(* IEC 61131-3 sources: AXOpen/src/components.rexroth.drives/ctrl/src/AxoCtrlxDriveXsc/v_6_x_x (part 2) *)

                        AxoStop_Deceleration := 1000.0;         // mm/s2
                        AxoStop_Jerk := 150000.0;               // mm/s3
                        AxoHalt_Deceleration := 1000.0;         // mm/s2
                        AxoHalt_Jerk := 150000.0;               // mm/s3
                        AxoHome_Position := 0.0;                // mm
                        AxoHome_HommingMode := 615;             // Negative direction, travel range limit switch, negative edge (NC contact), no Home switch evaluation, no Reference mark evaluation
                        AxoHome_Velocity := 2.0;                // mm/s
                        AxoHome_Acceleration := 1000.0;         // mm/s2
                        AxoHome_Deceleration := 1000.0;         // mm/s2
                        AxoSetPosition_Position := 0.0;         // mm
                        AxoMoveAbsolute_Position := 0.0;        // mm
                        AxoMoveAbsolute_Velocity := 5.0;        // mm/s
                        AxoMoveAbsolute_Acceleration := 1000.0; // mm/s2
                        AxoMoveAbsolute_Deceleration := 1000.0; // mm/s2
                        AxoMoveAbsolute_Jerk := 150000.0;       // mm/s3
                        AxoMoveRelative_Distance := 5.0;        // mm
                        AxoMoveRelative_Velocity := 5.0;        // mm/s
                        AxoMoveRelative_Acceleration := 1000.0; // mm/s2
                        AxoMoveRelative_Deceleration := 1000.0; // mm/s2
                        AxoMoveRelative_Jerk := 150000.0;       // mm/s3
                        AxoMoveAdditive_Distance := 5.0;        // mm
                        AxoMoveAdditive_Velocity := 5.0;        // mm/s
                        AxoMoveAdditive_Acceleration := 1000.0; // mm/s2
                        AxoMoveAdditive_Deceleration := 1000.0; // mm/s2
                        AxoMoveAdditive_Jerk := 150000.0;       // mm/s3
                        AxoMoveVelocity_Velocity := 5.0;        // mm/s
                        AxoMoveVelocity_Acceleration := 1000.0; // mm/s2
                        AxoMoveVelocity_Deceleration := 1000.0; // mm/s2
                        AxoMoveVelocity_Jerk := 150000.0;       // mm/s3
                        AxoTorqueControl_Torque := 0.0;         // N
                        AxoTorqueControl_TorqueRamp := 1.0;     // N/s
                        AxoTorqueControl_Velocity := 5.0;       // mm/s
                        AxoTorqueControl_Acceleration := 1000.0;// mm/s2
                        AxoTorqueControl_Deceleration := 1000.0;// mm/s2
                        AxoTorqueControl_Jerk := 150000.0;      // mm/s3
                        AxoJog_Velocity := 2.0;                 // mm/s
                        AxoJog_Acceleration := 500.0;           // mm/s2
                        AxoJog_Deceleration := 500.0;           // mm/s2
                        AxoJog_Jerk := 150000.0;                // mm/s3
                        AxisRefExt.Outputs.BipolarTorqueLimitation_S_0_0092_0_0 := INT#1000;  // 1000~~ 100%
                    ELSIF AxisType = eAxoDriveAxisType#Rotary THEN
                        //  Position
                        ScalingConstantRequiredPosition     :=  TO_LREAL(_S_0_0079) / LREAL#360.0;
                        ScalingConstantActualPosition       :=  LREAL#1.0/ScalingConstantRequiredPosition;
                        //  Velocity
                        ScalingConstantRequiredVelocity     := _exp[-_S_0_0046] / (TO_LREAL(_S_0_0045));
                        ScalingConstantActualVelocity       := LREAL#1.0/ScalingConstantRequiredVelocity;
                        //  Acceleration
                        ScalingConstantRequiredAcceleration :=  _exp[-_S_0_0162] / (TO_LREAL(_S_0_0161) * LREAL#180.0 /System.Math.Constants#PI);
                        ScalingConstantActualAcceleration   := LREAL#1.0/ScalingConstantRequiredAcceleration;
                        //  Deceleration
                        ScalingConstantRequiredDeceleration := ScalingConstantRequiredAcceleration;
                        ScalingConstantActualDeceleration   := ScalingConstantActualAcceleration;
                        //  Torque
                        ScalingConstantActualTorque         := TO_LREAL(_S_0_0093) *_exp[_S_0_0094];
                        ScalingConstantRequiredTorque       := LREAL#1.0/ScalingConstantActualTorque;
                        //  Jerk
                        ScalingConstantRequiredJerk         :=  ScalingConstantRequiredAcceleration;
                        ScalingConstantActualJerk           :=  LREAL#1.0/ScalingConstantRequiredJerk;

                        AxoStop_Deceleration := 36000.0;            // deg/s2
                        AxoStop_Jerk := 3600000.0;                  // deg/s3
                        AxoHalt_Deceleration := 36000.0;            // deg/s2
                        AxoHalt_Jerk := 3600000.0;                  // deg/s3
                        AxoHome_Position := 0.0;                    // deg
                        AxoHome_HommingMode := 71;                  // Negative direction, negative edge (NC contact), homing switch connected to drive, no Reference mark evaluation
                        AxoHome_Velocity := 45.0;                   // deg/s
                        AxoHome_Acceleration := 36000.0;            // deg/s2
                        AxoHome_Deceleration := 36000.0;            // deg/s2
                        AxoSetPosition_Position := 0.0;             // deg
                        AxoMoveAbsolute_Position := 0.0;            // deg
                        AxoMoveAbsolute_Velocity := 3600.0;         // deg/s
                        AxoMoveAbsolute_Acceleration := 36000.0;    // deg/s2
                        AxoMoveAbsolute_Deceleration := 36000.0;    // deg/s2
                        AxoMoveAbsolute_Jerk := 3600000.0;          // deg/s3
                        AxoMoveRelative_Distance := 360.0;          // deg
                        AxoMoveRelative_Velocity := 3600.0;         // deg/s
                        AxoMoveRelative_Acceleration := 36000.0;    // deg/s2
                        AxoMoveRelative_Deceleration := 36000.0;    // deg/s2
                        AxoMoveRelative_Jerk := 3600000.0;          // deg/s3
                        AxoMoveAdditive_Distance := 360.0;          // deg
                        AxoMoveAdditive_Velocity := 3600.0;         // deg/s
                        AxoMoveAdditive_Acceleration := 36000.0;    // deg/s2
                        AxoMoveAdditive_Deceleration := 36000.0;    // deg/s2
                        AxoMoveAdditive_Jerk := 3600000.0;          // deg/s3
                        AxoMoveVelocity_Velocity := 3600.0;         // deg/s
                        AxoMoveVelocity_Acceleration := 36000.0;    // deg/s2
                        AxoMoveVelocity_Deceleration := 36000.0;    // deg/s2
                        AxoMoveVelocity_Jerk := 3600000.0;          // deg/s3
                        AxoTorqueControl_Torque := 0.0;             // Nm
                        AxoTorqueControl_TorqueRamp := 1.0;         // Nm/s
                        AxoTorqueControl_Velocity := 3600.0;        // deg/s
                        AxoTorqueControl_Acceleration := 36000.0;   // deg/s2
                        AxoTorqueControl_Deceleration := 36000.0;   // deg/s2
                        AxoTorqueControl_Jerk := 3600000.0;         // deg/s3
                        AxoJog_Velocity := 45.0;                    // deg/s
                        AxoJog_Acceleration := 720.0;               // deg/s2
                        AxoJog_Deceleration := 720.0;               // deg/s2
                        AxoJog_Jerk := 1800000.0;                   // deg/s3
                        AxisRefExt.Outputs.BipolarTorqueLimitation_S_0_0092_0_0 := INT#1000;  // 1000~~ 100%
                    END_IF;
                    _ScalingRead := TRUE;
                    _State := UINT#50;
                END_IF;
                RETURN;
            END_IF;
            // Retrigger the reading of the scaling parameters in case of leaving the operation mode.
            IF (*_ScalingRead AND*) NOT AxisRefExt.Inputs.DriveStatusWord_S_0_0135_0_0.ReadyForOperationBit1 AND
                (AxisRefExt.Inputs.SignalStatusWord_S_0_0144_0_0.CmPmOmBit0 OR  AxisRefExt.Inputs.SignalStatusWord_S_0_0144_0_0.CmPmOmBit1 ) THEN
                _ScalingRead := FALSE;
                _State := UINT#0;
            END_IF;

            //*************************************************//

            Messenger.ActivateOnCondition(ULINT#300, Enable AND NOT EnablePositive, eAxoMessageCategory#Info);
            Messenger.ActivateOnCondition(ULINT#301, Enable AND NOT EnableNegative, eAxoMessageCategory#Info);

            //************************************************************
            SUPER.Run(THIS,AxisRefExt,Enable,EnablePositive,EnableNegative);
            //************************************************************

            THIS.ActualPosition := AxisRefExt.Inputs.ActualPosition_S_0_0386_0_0 * ScalingConstantActualPosition;
            THIS.ActualVelocity := AxisRefExt.Inputs.ActualVelocity_S_0_0535_0_0 * ScalingConstantActualVelocity;
            THIS.ActualTorque   := AxisRefExt.Inputs.ActualTorque_S_0_0084_0_0  * ScalingConstantActualTorque;

            IF NOT AxisRefExt.Inputs.DriveStatusWord_S_0_0135_0_0.ReadyForOperationBit0 THEN
                DriveState := AXOpen.Components.Drives.eAxoDriveState#Disabled;
            ELSIF _State>=UINT#310 AND _State<=UINT#327 AND
                    (NOT AxisRefExt.Inputs.DriveStatusWord_S_0_0135_0_0.InReference OR NOT AxisRefExt.Inputs.DriveStatusWord_S_0_0135_0_0.InStandstill ) THEN
                DriveState := AXOpen.Components.Drives.eAxoDriveState#Homing;
            ELSIF   _State>=UINT#350 AND _State<=UINT#357 OR                                            //******MC_MoveAbsolute***************
                    _State>=UINT#360 AND _State<=UINT#367 OR                                            //******MC_MoveRelative***************
                    _State>=UINT#370 AND _State<=UINT#377 THEN                                          //******MC_MoveAditive****************
                DriveState := AXOpen.Components.Drives.eAxoDriveState#DiscreteMotion;
            ELSIF (_State>=UINT#380 AND _State<UINT#387) OR                                             //(************************************
                    AxisRefExt.Outputs.SignalControlWord_S_0_0145_0_0.JogNegative OR                    //******MC_MoveVelocity OR MC_Jog******
                    AxisRefExt.Outputs.SignalControlWord_S_0_0145_0_0.JogPositive OR                    //************************************)
                    _State>=UINT#390 AND _State<UINT#397 OR                                             //(************************************
                    (   AxisRefExt.Inputs.DriveStatusWord_S_0_0135_0_0.ActualOperatingModeBit0 AND      //*************************************
                    NOT AxisRefExt.Inputs.DriveStatusWord_S_0_0135_0_0.ActualOperatingModeBit1 AND      //******MC_TorqueControl***************
                    NOT AxisRefExt.Inputs.DriveStatusWord_S_0_0135_0_0.ActualOperatingModeBit2 AND      //*************************************
                        AxisRefExt.Outputs.DriveControlWord_S_0_0134_0_0.DriveHalt) THEN                //************************************)
                DriveState := AXOpen.Components.Drives.eAxoDriveState#ContinuousMotion;
            ELSIF FALSE THEN
                DriveState := AXOpen.Components.Drives.eAxoDriveState#SynchronizedMotion;               //*****Not implemented*****************
            ELSIF   AxisRefExt.Inputs.DriveStatusWord_S_0_0135_0_0.ReadyForOperationBit0 AND
                    AxisRefExt.Inputs.DriveStatusWord_S_0_0135_0_0.ReadyForOperationBit1 AND
                    NOT AxisRefExt.Outputs.DriveControlWord_S_0_0134_0_0.DriveHalt AND
                    NOT AxisRefExt.Inputs.DriveStatusWord_S_0_0135_0_0.InStandstill THEN
                DriveState := AXOpen.Components.Drives.eAxoDriveState#Stopping;
            ELSIF AxisRefExt.Inputs.DriveStatusWord_S_0_0135_0_0.DriveErrorZKL1 THEN
                DriveState := AXOpen.Components.Drives.eAxoDriveState#Errorstop;
            ELSIF AxisRefExt.Inputs.DriveStatusWord_S_0_0135_0_0.InStandstill THEN
                DriveState := AXOpen.Components.Drives.eAxoDriveState#Standstill;
            END_IF;

            Messenger.ActivateOnCondition(THIS.MessageCodeFromMC, THIS.ErrorFromMC AND MessageCodeFromMC = _lastMessageCodeFromMC ,eAxoMessageCategory#Error);
            IF Messenger.MessengerState = eAxoMessengerState#Idle THEN
                IF THIS.ErrorFromMC THEN
                    _lastMessageCodeFromMC := THIS.MessageCodeFromMC;
                ELSE
                    THIS.MessageCodeFromMC := ULINT#0;
                END_IF;
            END_IF;

            THIS.ErrorOutOfMC := NOT THIS.ErrorFromMC AND (AxisRefExt.Inputs.DriveStatusWord_S_0_0135_0_0.DriveErrorZKL1 OR (AxisRefExt.Inputs.DriveStatusWord_S_0_0135_0_0.WarningZKL2 AND AxisRefExt.Inputs.DiagnosticMessage_S_0_0390_0_0 >= DWORD#16#C00E0000));
            MessageCodeOutOfMC := TO_ULINT(AxisRefExt.Inputs.DiagnosticMessage_S_0_0390_0_0 AND DWORD#16#000FFFFF);
            Messenger.ActivateOnCondition(THIS.MessageCodeOutOfMC, THIS.ErrorOutOfMC AND MessageCodeOutOfMC = _lastMessageCodeOutOfMC ,eAxoMessageCategory#Error);
            IF Messenger.MessengerState = eAxoMessengerState#Idle THEN
                IF THIS.ErrorOutOfMC THEN
                    _lastMessageCodeOutOfMC := THIS.MessageCodeOutOfMC;
                ELSE
                    THIS.MessageCodeOutOfMC := ULINT#0;
                END_IF;
            END_IF;

            IF _ScalingRead AND _State = UINT#50 THEN
                // AxisRefExt.Outputs.SignalControlWord_S_0_0145_0_0.AcceptanceOfPositioningCommandValue := AxisRefExt.Inputs.SignalStatusWord_S_0_0144_0_0.PositionCommandAck;
                // THIS.AxoReset_Task.RemoteInvoke := TRUE;
                _State := UINT#0;
            END_IF;
        END_METHOD

        ///<summary>
        /// Ensures swapping the hardware input data structure into the AxisRef data structure
        ///</summary>
        METHOD PROTECTED  OVERRIDE UpdateInputs : BOOL
            VAR_INPUT
                AxisRef         :   AXOpen.Components.Abstractions.Drives.IAxoAxisReference;
            END_VAR
            VAR
                _AxisReference :  REF_TO AxoCtrlxDriveXscAxisReference;
            END_VAR

           _AxisReference ?= AxisRef;

           IF(_AxisReference = NULL) THEN
               Messenger.Activate(     UINT#1410, eAxoMessageCategory#ProgrammingError);
               DriveStatus.Error.Id := UINT#1410;
               RETURN;
           END_IF;

           _retVal := Siemens.Simatic.DistributedIO.ReadData((AxisRefExt.HWIDs.HW_S_0_0135_0_0) ,_data2);
           IF _retVal > WORD#0 THEN
               Messenger.Activate(     UINT#1201, eAxoMessageCategory#Error);
               DriveStatus.Error.Id := UINT#1201;
               RETURN;
           END_IF;

           AxisRefExt.Inputs.DriveStatusWord_S_0_0135_0_0._bit00_Reserve 			:=  _data2[1].%X0;     //  0
           AxisRefExt.Inputs.DriveStatusWord_S_0_0135_0_0._bit01_Reserve 			:=  _data2[1].%X1;     //  1
           AxisRefExt.Inputs.DriveStatusWord_S_0_0135_0_0._bit02_Reserve 			:=  _data2[1].%X2;     //  2
           AxisRefExt.Inputs.DriveStatusWord_S_0_0135_0_0.CommandProcessingStatus	:=  _data2[1].%X3;     //  3
           AxisRefExt.Inputs.DriveStatusWord_S_0_0135_0_0.InStandstill 			    :=  _data2[1].%X4;     //  4
           AxisRefExt.Inputs.DriveStatusWord_S_0_0135_0_0.InReference 			    :=  _data2[1].%X5;     //  5
           AxisRefExt.Inputs.DriveStatusWord_S_0_0135_0_0._bit06_Reserve 			:=  _data2[1].%X6;     //  6
           AxisRefExt.Inputs.DriveStatusWord_S_0_0135_0_0.HardwareLock              :=  _data2[1].%X7;     //  7
           AxisRefExt.Inputs.DriveStatusWord_S_0_0135_0_0.ActualOperatingModeBit0   :=  _data2[0].%X0;     //  8
           AxisRefExt.Inputs.DriveStatusWord_S_0_0135_0_0.ActualOperatingModeBit1   :=  _data2[0].%X1;     //  9
           AxisRefExt.Inputs.DriveStatusWord_S_0_0135_0_0.ActualOperatingModeBit2   :=  _data2[0].%X2;     //  10
           AxisRefExt.Inputs.DriveStatusWord_S_0_0135_0_0._bit11_Reserve 			:=  _data2[0].%X3;     //  11
           AxisRefExt.Inputs.DriveStatusWord_S_0_0135_0_0.WarningZKL2 			    :=  _data2[0].%X4;     //  12
           AxisRefExt.Inputs.DriveStatusWord_S_0_0135_0_0.DriveErrorZKL1 			:=  _data2[0].%X5;     //  13
           AxisRefExt.Inputs.DriveStatusWord_S_0_0135_0_0.ReadyForOperationBit0     :=  _data2[0].%X6;     //  14
           AxisRefExt.Inputs.DriveStatusWord_S_0_0135_0_0.ReadyForOperationBit1     :=  _data2[0].%X7;     //  15

           _retVal := Siemens.Simatic.DistributedIO.ReadData((AxisRefExt.HWIDs.HW_S_0_0144_0_0) ,_data2);
           IF _retVal > WORD#0 THEN
               Messenger.Activate(     UINT#1202, eAxoMessageCategory#Error);
               DriveStatus.Error.Id := UINT#1202;
               RETURN;
           END_IF;

           AxisRefExt.Inputs.SignalStatusWord_S_0_0144_0_0.CmPmOmBit0 			    :=  _data2[1].%X0;     //  0
           AxisRefExt.Inputs.SignalStatusWord_S_0_0144_0_0.CmPmOmBit1 			    :=  _data2[1].%X1;     //  1
           AxisRefExt.Inputs.SignalStatusWord_S_0_0144_0_0.InTargetPosition 	    :=  _data2[1].%X2;     //  2
           AxisRefExt.Inputs.SignalStatusWord_S_0_0144_0_0.PositionCommandAck	    :=  _data2[1].%X3;     //  3
           AxisRefExt.Inputs.SignalStatusWord_S_0_0144_0_0.DriveStandstill 	        :=  _data2[1].%X4;     //  4
           AxisRefExt.Inputs.SignalStatusWord_S_0_0144_0_0.CommandChangeBit 	    :=  _data2[1].%X5;     //  5
           AxisRefExt.Inputs.SignalStatusWord_S_0_0144_0_0._bit6_Reserve 			:=  _data2[1].%X6;     //  6
           AxisRefExt.Inputs.SignalStatusWord_S_0_0144_0_0._bit7_Reserve            :=  _data2[1].%X7;     //  7
           AxisRefExt.Inputs.SignalStatusWord_S_0_0144_0_0.LockedByHardware         :=  _data2[0].%X0;     //  8
           AxisRefExt.Inputs.SignalStatusWord_S_0_0144_0_0._bit9_Reserve            :=  _data2[0].%X1;     //  9
           AxisRefExt.Inputs.SignalStatusWord_S_0_0144_0_0._bit10_Reserve           :=  _data2[0].%X2;     //  10
           AxisRefExt.Inputs.SignalStatusWord_S_0_0144_0_0._bit11_Reserve 			:=  _data2[0].%X3;     //  11
           AxisRefExt.Inputs.SignalStatusWord_S_0_0144_0_0._bit12_Reserve 			:=  _data2[0].%X4;     //  12
           AxisRefExt.Inputs.SignalStatusWord_S_0_0144_0_0._bit13_Reserve 			:=  _data2[0].%X5;     //  13
           AxisRefExt.Inputs.SignalStatusWord_S_0_0144_0_0._bit14_Reserve           :=  _data2[0].%X6;     //  14
           AxisRefExt.Inputs.SignalStatusWord_S_0_0144_0_0._bit15_Reserve           :=  _data2[0].%X7;     //  15

           _retVal := Siemens.Simatic.DistributedIO.ReadData((AxisRefExt.HWIDs.HW_S_0_0386_0_0) ,_data4);
           IF _retVal > WORD#0 THEN
               Messenger.Activate(     UINT#1203, eAxoMessageCategory#Error);
               DriveStatus.Error.Id := UINT#1203;
               RETURN;
           END_IF;
           _dword.%B3  :=  _data4[0];
           _dword.%B2  :=  _data4[1];
           _dword.%B1  :=  _data4[2];
           _dword.%B0  :=  _data4[3];
           AxisRefExt.Inputs.ActualPosition_S_0_0386_0_0 := TO_DINT(_dword);

           _retVal := Siemens.Simatic.DistributedIO.ReadData((AxisRefExt.HWIDs.HW_S_0_0535_0_0) ,_data4);
           IF _retVal > WORD#0 THEN
               Messenger.Activate(     UINT#1204, eAxoMessageCategory#Error);
               DriveStatus.Error.Id := UINT#1204;
               RETURN;
           END_IF;
           _dword.%B3  :=  _data4[0];
           _dword.%B2  :=  _data4[1];
           _dword.%B1  :=  _data4[2];
           _dword.%B0  :=  _data4[3];
           AxisRefExt.Inputs.ActualVelocity_S_0_0535_0_0 := TO_DINT(_dword);

           _retVal := Siemens.Simatic.DistributedIO.ReadData((AxisRefExt.HWIDs.HW_S_0_0390_0_0) ,_data4);
           IF _retVal > WORD#0 THEN
               Messenger.Activate(     UINT#1205, eAxoMessageCategory#Error);
               DriveStatus.Error.Id := UINT#1205;
               RETURN;
           END_IF;
           _dword.%B3  :=  _data4[0];
           _dword.%B2  :=  _data4[1];
           _dword.%B1  :=  _data4[2];
           _dword.%B0  :=  _data4[3];
           AxisRefExt.Inputs.DiagnosticMessage_S_0_0390_0_0 := _dword;

           _retVal := Siemens.Simatic.DistributedIO.ReadData((AxisRefExt.HWIDs.HW_S_0_1720_0_2) ,_data2);
           IF _retVal > WORD#0 THEN
               Messenger.Activate(     UINT#1206, eAxoMessageCategory#Error);
               DriveStatus.Error.Id := UINT#1206;
               RETURN;
           END_IF;
           AxisRefExt.Inputs.SupplyUnitStatusWord_S_0_1720_0_2._bit0_Reserve 				        := _data2[1].%X0;
           AxisRefExt.Inputs.SupplyUnitStatusWord_S_0_1720_0_2._bit1_Reserve 				        := _data2[1].%X1;
           AxisRefExt.Inputs.SupplyUnitStatusWord_S_0_1720_0_2._bit2_Reserve 				        := _data2[1].%X2;
           AxisRefExt.Inputs.SupplyUnitStatusWord_S_0_1720_0_2._bit3_Reserve 				        := _data2[1].%X3;
           AxisRefExt.Inputs.SupplyUnitStatusWord_S_0_1720_0_2.MainsStatus				            := _data2[1].%X4;
           AxisRefExt.Inputs.SupplyUnitStatusWord_S_0_1720_0_2.HardwareEnable				        := _data2[1].%X5;
           AxisRefExt.Inputs.SupplyUnitStatusWord_S_0_1720_0_2.ControllingTheMainsConnection        := _data2[1].%X6;
           AxisRefExt.Inputs.SupplyUnitStatusWord_S_0_1720_0_2.BbContact				            := _data2[1].%X7;
           AxisRefExt.Inputs.SupplyUnitStatusWord_S_0_1720_0_2.PreselectedOPmodesFB_bit0            := _data2[0].%X0;
           AxisRefExt.Inputs.SupplyUnitStatusWord_S_0_1720_0_2.PreselectedOPmodesFB_bit01           := _data2[0].%X1;
           AxisRefExt.Inputs.SupplyUnitStatusWord_S_0_1720_0_2.DCbusDischarge                       := _data2[0].%X2;
           AxisRefExt.Inputs.SupplyUnitStatusWord_S_0_1720_0_2.BrakingResistor                      := _data2[0].%X3;
           AxisRefExt.Inputs.SupplyUnitStatusWord_S_0_1720_0_2.Warning                              := _data2[0].%X4;
           AxisRefExt.Inputs.SupplyUnitStatusWord_S_0_1720_0_2.Error                                := _data2[0].%X5;
           AxisRefExt.Inputs.SupplyUnitStatusWord_S_0_1720_0_2.ReadyForEnabling                     := _data2[0].%X6;
           AxisRefExt.Inputs.SupplyUnitStatusWord_S_0_1720_0_2.Enabling                             := _data2[0].%X7;

           _retVal := Siemens.Simatic.DistributedIO.ReadData((AxisRefExt.HWIDs.HW_S_0_0084_0_0) ,_data2);
           IF _retVal > WORD#0 THEN
               Messenger.Activate(     UINT#1207, eAxoMessageCategory#Error);
               DriveStatus.Error.Id := UINT#1207;
               RETURN;
           END_IF;
           _word.%B1  :=  _data2[0];
           _word.%B0  :=  _data2[1];
           AxisRefExt.Inputs.ActualTorque_S_0_0084_0_0 := TO_INT(_word);
        END_METHOD

        ///<summary>
        /// Ensures swapping the AxisRef data structure into the hardware output data structure
        ///</summary>
        METHOD PROTECTED OVERRIDE UpdateOutputs : BOOL
            VAR_INPUT
                AxisRef         :   AXOpen.Components.Abstractions.Drives.IAxoAxisReference;
            END_VAR
            VAR
                _AxisReference :  REF_TO AxoCtrlxDriveXscAxisReference;
            END_VAR
            _AxisReference ?= AxisRef;

            IF(_AxisReference = NULL) THEN
                Messenger.Activate(     UINT#1420, eAxoMessageCategory#ProgrammingError);
                DriveStatus.Error.Id := UINT#1420;
                RETURN;
            END_IF;
            //***********Update outputs **************
            _data2[1].%X0   :=  AxisRefExt.Outputs.DriveControlWord_S_0_0134_0_0._bit00_Reserve;
            _data2[1].%X1   :=  AxisRefExt.Outputs.DriveControlWord_S_0_0134_0_0._bit01_Reserve;
            _data2[1].%X2   :=  AxisRefExt.Outputs.DriveControlWord_S_0_0134_0_0._bit02_Reserve;
            _data2[1].%X3   :=  AxisRefExt.Outputs.DriveControlWord_S_0_0134_0_0._bit03_Reserve;
            _data2[1].%X4   :=  AxisRefExt.Outputs.DriveControlWord_S_0_0134_0_0._bit04_Reserve;
            _data2[1].%X5   :=  AxisRefExt.Outputs.DriveControlWord_S_0_0134_0_0._bit05_Reserve;
            _data2[1].%X6   :=  AxisRefExt.Outputs.DriveControlWord_S_0_0134_0_0._bit06_Reserve;
            _data2[1].%X7   :=  AxisRefExt.Outputs.DriveControlWord_S_0_0134_0_0._bit07_Reserve;
            _data2[0].%X0   :=  AxisRefExt.Outputs.DriveControlWord_S_0_0134_0_0.CommandOperationModeBit0;
            _data2[0].%X1   :=  AxisRefExt.Outputs.DriveControlWord_S_0_0134_0_0.CommandOperationModeBit1;
            _data2[0].%X2   :=  AxisRefExt.Outputs.DriveControlWord_S_0_0134_0_0.CommandOperationModeBit2;
            _data2[0].%X3   :=  AxisRefExt.Outputs.DriveControlWord_S_0_0134_0_0._bit11_Reserve;
            _data2[0].%X4   :=  AxisRefExt.Outputs.DriveControlWord_S_0_0134_0_0._bit12_Reserve;
            _data2[0].%X5   :=  AxisRefExt.Outputs.DriveControlWord_S_0_0134_0_0.DriveHalt;
            _data2[0].%X6   :=  AxisRefExt.Outputs.DriveControlWord_S_0_0134_0_0.DriveEnable;
            _data2[0].%X7   :=  AxisRefExt.Outputs.DriveControlWord_S_0_0134_0_0.DriveOn;

            _retVal := Siemens.Simatic.DistributedIO.WriteData((AxisRefExt.HWIDs.HW_S_0_0134_0_0),_data2);
            IF _retVal > WORD#0 THEN
                Messenger.Activate(     UINT#1231, eAxoMessageCategory#Error);
                DriveStatus.Error.Id := UINT#1231;
                RETURN;
            END_IF;

            _data2[1].%X0   :=  AxisRefExt.Outputs.SignalControlWord_S_0_0145_0_0.AcceptanceOfPositioningCommandValue;
            _data2[1].%X2   :=  AxisRefExt.Outputs.SignalControlWord_S_0_0145_0_0.HomingControl;
            _data2[1].%X3   :=  AxisRefExt.Outputs.SignalControlWord_S_0_0145_0_0.AbsoluteRelative;
            _data2[1].%X4   :=  AxisRefExt.Outputs.SignalControlWord_S_0_0145_0_0.ImmediateChange;
            _data2[1].%X5   :=  AxisRefExt.Outputs.SignalControlWord_S_0_0145_0_0.ClearError;
            _data2[1].%X6   :=  AxisRefExt.Outputs.SignalControlWord_S_0_0145_0_0.JogPositive;
            _data2[1].%X7   :=  AxisRefExt.Outputs.SignalControlWord_S_0_0145_0_0.JogNegative;
            _data2[0].%X0   :=  AxisRefExt.Outputs.SignalControlWord_S_0_0145_0_0.SwitchToCM;
            _data2[0].%X1   :=  AxisRefExt.Outputs.SignalControlWord_S_0_0145_0_0.SwitchTo0M;
            _data2[0].%X2   :=  AxisRefExt.Outputs.SignalControlWord_S_0_0145_0_0.CancelReferencePoint;
            _data2[0].%X3   :=  AxisRefExt.Outputs.SignalControlWord_S_0_0145_0_0.DeviceReboot;
            _data2[0].%X4   :=  AxisRefExt.Outputs.SignalControlWord_S_0_0145_0_0._bit12_Reserve;
            _data2[0].%X5   :=  AxisRefExt.Outputs.SignalControlWord_S_0_0145_0_0._bit13_Reserve;
            _data2[0].%X6   :=  AxisRefExt.Outputs.SignalControlWord_S_0_0145_0_0._bit14_Reserve;
            _data2[0].%X7   :=  AxisRefExt.Outputs.SignalControlWord_S_0_0145_0_0.SetAbsPositionFunction;

            _retVal := Siemens.Simatic.DistributedIO.WriteData((AxisRefExt.HWIDs.HW_S_0_0145_0_0),_data2);
            IF _retVal > WORD#0 THEN
                Messenger.Activate(     UINT#1232, eAxoMessageCategory#Error);
                DriveStatus.Error.Id := UINT#1232;
                RETURN;
            END_IF;

            _data4[3]   :=  AxisRefExt.Outputs.CommandPosition_S_0_0282_0_0.%B0;
            _data4[2]   :=  AxisRefExt.Outputs.CommandPosition_S_0_0282_0_0.%B1;
            _data4[1]   :=  AxisRefExt.Outputs.CommandPosition_S_0_0282_0_0.%B2;
            _data4[0]   :=  AxisRefExt.Outputs.CommandPosition_S_0_0282_0_0.%B3;

            _retVal := Siemens.Simatic.DistributedIO.WriteData((AxisRefExt.HWIDs.HW_S_0_0282_0_0),_data4);
            IF _retVal > WORD#0 THEN
                Messenger.Activate(     UINT#1233, eAxoMessageCategory#Error);
                DriveStatus.Error.Id := UINT#1233;
                RETURN;
            END_IF;

            _data4[3]   :=  AxisRefExt.Outputs.CommandVelocity_S_0_0259_0_0.%B0;
            _data4[2]   :=  AxisRefExt.Outputs.CommandVelocity_S_0_0259_0_0.%B1;
            _data4[1]   :=  AxisRefExt.Outputs.CommandVelocity_S_0_0259_0_0.%B2;
            _data4[0]   :=  AxisRefExt.Outputs.CommandVelocity_S_0_0259_0_0.%B3;

            _retVal := Siemens.Simatic.DistributedIO.WriteData((AxisRefExt.HWIDs.HW_S_0_0259_0_0),_data4);
            IF _retVal > WORD#0 THEN
                Messenger.Activate(     UINT#1234, eAxoMessageCategory#Error);
                DriveStatus.Error.Id := UINT#1234;
                RETURN;
            END_IF;

            _data4[3]   :=  AxisRefExt.Outputs.CommandAcceleration_S_0_0260_0_0.%B0;
            _data4[2]   :=  AxisRefExt.Outputs.CommandAcceleration_S_0_0260_0_0.%B1;
            _data4[1]   :=  AxisRefExt.Outputs.CommandAcceleration_S_0_0260_0_0.%B2;
            _data4[0]   :=  AxisRefExt.Outputs.CommandAcceleration_S_0_0260_0_0.%B3;

            _retVal := Siemens.Simatic.DistributedIO.WriteData((AxisRefExt.HWIDs.HW_S_0_0260_0_0),_data4);
            IF _retVal > WORD#0 THEN
                Messenger.Activate(     UINT#1235, eAxoMessageCategory#Error);
                DriveStatus.Error.Id := UINT#1235;
                RETURN;
            END_IF;

            _data4[3]   :=  AxisRefExt.Outputs.CommandDecceleration_S_0_0359_0_0.%B0;
            _data4[2]   :=  AxisRefExt.Outputs.CommandDecceleration_S_0_0359_0_0.%B1;
            _data4[1]   :=  AxisRefExt.Outputs.CommandDecceleration_S_0_0359_0_0.%B2;
            _data4[0]   :=  AxisRefExt.Outputs.CommandDecceleration_S_0_0359_0_0.%B3;

            _retVal := Siemens.Simatic.DistributedIO.WriteData((AxisRefExt.HWIDs.HW_S_0_0359_0_0),_data4);
            IF _retVal > WORD#0 THEN
                Messenger.Activate(     UINT#1236, eAxoMessageCategory#Error);
                DriveStatus.Error.Id := UINT#1236;
                RETURN;
            END_IF;

            _data2[1].%X0   :=  AxisRefExt.Outputs.SupplyUnitControlWord_S_0_1720_0_1._bit0_Reserve;
            _data2[1].%X1   :=  AxisRefExt.Outputs.SupplyUnitControlWord_S_0_1720_0_1._bit1_Reserve;
            _data2[1].%X2   :=  AxisRefExt.Outputs.SupplyUnitControlWord_S_0_1720_0_1._bit2_Reserve;
            _data2[1].%X3   :=  AxisRefExt.Outputs.SupplyUnitControlWord_S_0_1720_0_1._bit3_Reserve;
            _data2[1].%X4   :=  AxisRefExt.Outputs.SupplyUnitControlWord_S_0_1720_0_1._bit4_Reserve;
            _data2[1].%X5   :=  AxisRefExt.Outputs.SupplyUnitControlWord_S_0_1720_0_1._bit5_Reserve;
            _data2[1].%X6   :=  AxisRefExt.Outputs.SupplyUnitControlWord_S_0_1720_0_1._bit6_Reserve;
            _data2[1].%X7   :=  AxisRefExt.Outputs.SupplyUnitControlWord_S_0_1720_0_1._bit7_Reserve;
            _data2[0].%X0   :=  AxisRefExt.Outputs.SupplyUnitControlWord_S_0_1720_0_1.ModeSelectionBit0;
            _data2[0].%X1   :=  AxisRefExt.Outputs.SupplyUnitControlWord_S_0_1720_0_1.ModeSelectionBit1;
            _data2[0].%X2   :=  AxisRefExt.Outputs.SupplyUnitControlWord_S_0_1720_0_1.DCbusDischarge;
            _data2[0].%X3   :=  AxisRefExt.Outputs.SupplyUnitControlWord_S_0_1720_0_1._bit11_Reserve;
            _data2[0].%X4   :=  AxisRefExt.Outputs.SupplyUnitControlWord_S_0_1720_0_1.ControllingTheReadyForOperationRelay;
            _data2[0].%X5   :=  AxisRefExt.Outputs.SupplyUnitControlWord_S_0_1720_0_1._bit13_Reserve;
            _data2[0].%X6   :=  AxisRefExt.Outputs.SupplyUnitControlWord_S_0_1720_0_1.ControllingDCbusChargingAndMainsContactor;
            _data2[0].%X7   :=  AxisRefExt.Outputs.SupplyUnitControlWord_S_0_1720_0_1.Enabling;

            _retVal := Siemens.Simatic.DistributedIO.WriteData((AxisRefExt.HWIDs.HW_S_0_1720_0_1),_data2);
            IF _retVal > WORD#0 THEN
                Messenger.Activate(     UINT#1237, eAxoMessageCategory#Error);
                DriveStatus.Error.Id := UINT#1237;
                RETURN;
            END_IF;

            _data2[1]   :=  AxisRefExt.Outputs.BipolarTorqueLimitation_S_0_0092_0_0.%B0;
            _data2[0]   :=  AxisRefExt.Outputs.BipolarTorqueLimitation_S_0_0092_0_0.%B1;

            _retVal := Siemens.Simatic.DistributedIO.WriteData((AxisRefExt.HWIDs.HW_S_0_0092_0_0),_data2);
            IF _retVal > WORD#0 THEN
                Messenger.Activate(     UINT#1238, eAxoMessageCategory#Error);
                DriveStatus.Error.Id := UINT#1238;
                RETURN;
            END_IF;

            _data2[1]   :=  AxisRefExt.Outputs.CommandTorque_S_0_0080_0_0.%B0;
            _data2[0]   :=  AxisRefExt.Outputs.CommandTorque_S_0_0080_0_0.%B1;

            _retVal := Siemens.Simatic.DistributedIO.WriteData((AxisRefExt.HWIDs.HW_S_0_0080_0_0),_data2);
            IF _retVal > WORD#0 THEN
                Messenger.Activate(     UINT#1239, eAxoMessageCategory#Error);
                DriveStatus.Error.Id := UINT#1239;
                RETURN;
            END_IF;

            _data4[3]   :=  AxisRefExt.Outputs.CommandJerk_S_0_0193_0_0.%B0;
            _data4[2]   :=  AxisRefExt.Outputs.CommandJerk_S_0_0193_0_0.%B1;
            _data4[1]   :=  AxisRefExt.Outputs.CommandJerk_S_0_0193_0_0.%B2;
            _data4[0]   :=  AxisRefExt.Outputs.CommandJerk_S_0_0193_0_0.%B3;

            _retVal := Siemens.Simatic.DistributedIO.WriteData((AxisRefExt.HWIDs.HW_S_0_0193_0_0),_data4);
            IF _retVal > WORD#0 THEN
                Messenger.Activate(     UINT#1240, eAxoMessageCategory#Error);
                DriveStatus.Error.Id := UINT#1240;
                RETURN;
            END_IF;

            //************************************************************

        END_METHOD

        ///<summary>
        /// This method controls the power stage (On or Off).
        ///</summary>
        VAR INTERNAL
            MC_PowerEnable_PV					:	BOOL := FALSE;		//Enable - previous value
            MC_PowerErrorID					    : 	DINT;
        END_VAR
        METHOD PUBLIC OVERRIDE MC_Power
            VAR_INPUT
                AxisRef         :   AXOpen.Components.Abstractions.Drives.IAxoAxisReference;
                Enable          :   BOOL;                       //  As long as ‘Enable’ is true, power is being enabled.
            END_VAR
            VAR_OUTPUT
                Status          :   BOOL;                       //  Effective_State of the power stage
                Valid           :   BOOL;                       //  If true, a valid set of outputs is available at the method
                Error           :   BOOL;                       //  Signals that an error has occurred within the method
                ErrorID         :   DINT;                       //  Error identification
            END_VAR
            VAR
                _AxisReference :  REF_TO AxoCtrlxDriveXscAxisReference;
            END_VAR

            _AxisReference ?= AxisRef;

            IF(_AxisReference = NULL) THEN
                Messenger.Activate(     UINT#1430, eAxoMessageCategory#Error);
                DriveStatus.Error.Id := UINT#1430;
                RETURN;
            END_IF;

            Valid   := FALSE;
            IF Enable THEN
                IF NOT MC_PowerEnable_PV THEN
                    _AxisReference^.Outputs.DriveControlWord_S_0_0134_0_0.DriveEnable   :=  TRUE;
                    _AxisReference^.Outputs.DriveControlWord_S_0_0134_0_0.DriveOn       :=  TRUE;
                END_IF;
                IF NOT  _AxisReference^.Inputs.DriveStatusWord_S_0_0135_0_0.DriveErrorZKL1 AND
                        _AxisReference^.Inputs.DriveStatusWord_S_0_0135_0_0.ReadyForOperationBit0 AND
                        _AxisReference^.Inputs.DriveStatusWord_S_0_0135_0_0.ReadyForOperationBit1 THEN
                    Status  := TRUE;
                    Valid   := TRUE;
                ELSE
                    Status  := FALSE;
                    Valid   := TRUE;
                END_IF;
                // IF _AxisReference^.Inputs.DriveStatusWord_S_0_0135_0_0.DriveErrorZKL1 OR (_AxisReference^.Inputs.DriveStatusWord_S_0_0135_0_0.WarningZKL2 AND _AxisReference^.Inputs.DiagnosticMessage_S_0_0390_0_0 >= DWORD#16#C00E0000) THEN
                IF _AxisReference^.Inputs.DriveStatusWord_S_0_0135_0_0.DriveErrorZKL1 AND (NOT _AxisReference^.Inputs.DriveStatusWord_S_0_0135_0_0.ReadyForOperationBit0 OR NOT _AxisReference^.Inputs.DriveStatusWord_S_0_0135_0_0.ReadyForOperationBit1) THEN
                    Status	:= FALSE;
                    Error   := TRUE;
                    MC_PowerErrorID := TO_DINT(_AxisReference^.Inputs.DiagnosticMessage_S_0_0390_0_0 AND DWORD#16#000FFFFF);
                END_IF;
            END_IF;

            IF NOT Enable AND MC_PowerEnable_PV THEN
                MC_PowerErrorID := DINT#0;
                _AxisReference^.Outputs.DriveControlWord_S_0_0134_0_0.DriveEnable   :=  FALSE;
                _AxisReference^.Outputs.DriveControlWord_S_0_0134_0_0.DriveOn       :=  FALSE;
            END_IF;

            ErrorID := MC_PowerErrorID;
            MC_PowerEnable_PV := Enable;
        END_METHOD

        ///<summary>
        /// This method commands the axis to perform the «search home» sequence. The details of this sequence are
        /// manufacturer dependent and can be set by the axis’ parameters. The ‘Position’ input is used to set the absolute
        /// position when reference signal is detected. This method completes at ‘Standstill’ if it was started in ‘Standstill’.
        ///</summary>
        VAR INTERNAL
            MC_HomeExecute_PV					: 	BOOL;				//Execute - previous value
            MC_HomeErrorID					    : 	DINT;
            MC_HomeCycle					    : 	ULINT;
        END_VAR
        METHOD PUBLIC OVERRIDE MC_Home
            VAR_INPUT
                AxisRef         :   AXOpen.Components.Abstractions.Drives.IAxoAxisReference;
                Execute         :   BOOL;                       //  Start the motion at rising edge
                Position        :   LREAL;                      //  Absolute position when the reference signal is detected
                HommingMode     :   INT;                        //  Required homming mode
                Velocity        :   LREAL;                      //  Value of the maximum ‘Velocity’ (not necessarily reached) [u/s].
                Acceleration    :   LREAL;                      //  Value of the ‘Acceleration’ (always positive) (increasing energy of the motor) [u/s2]
                Deceleration    :   LREAL;                      //  Value of the ‘Deceleration’ (always positive) (decreasing energy of the motor) [u/s2]
            END_VAR
            VAR_OUTPUT
                Done            :   BOOL;                       // Reference known and set sucessfully
                Busy            :   BOOL;                       // The method is not finished and new output values are to be expected
                Active          :   BOOL;                       // Indicates that the method has control on the axis
                CommandAborted  :   BOOL;                       // ‘Command’ is aborted by another command
                Error           :   BOOL;                       // Signals that an error has occurred within the method
                ErrorID         :   DINT;                       // Error identification
             END_VAR
             VAR
                _AxisReference :  REF_TO AxoCtrlxDriveXscAxisReference;
            END_VAR

            _AxisReference ?= AxisRef;

            IF(_AxisReference = NULL) THEN
                Messenger.Activate(     UINT#1440, eAxoMessageCategory#ProgrammingError);
                DriveStatus.Error.Id := UINT#1440;
                RETURN;
            END_IF;

            IF THIS.AxoHome_Task.StartTriggered() THEN
                _AxisReference^.Status.CurrentMotionTaskId := AXOpen.Components.Drives.eAxoMotionTaskId#Axo_Home;
            END_IF;

            IF Execute AND NOT MC_HomeExecute_PV AND _State = UINT#0 THEN
                _AxisReference^.Data.Cycle := _AxisReference^.Data.Cycle + ULINT#2;
                MC_HomeCycle := _AxisReference^.Data.Cycle ;
            END_IF;

            IF Execute THEN
                Messenger.ActivateOnCondition(ULINT#1441, Execute AND Acceleration <= 0, eAxoMessageCategory#ProgrammingError);
                Messenger.ActivateOnCondition(ULINT#1442, Execute AND Deceleration <= 0, eAxoMessageCategory#ProgrammingError);

                IF _State = UINT#0 THEN
                    Busy := TRUE;
                    Active := TRUE;
                    MC_HomeErrorID :=  DINT#0;
                    DriveStatus.Error.Id :=  UINT#0;
                    TaskMessenger.Restore();
                    _tmpTimer.OnDelay(THIS, FALSE , T#0s);
                    // _AxisReference^.Outputs.DriveControlWord_S_0_0134_0_0.IPOSYNC := FALSE;
                    // _AxisReference^.Outputs.DriveControlWord_S_0_0134_0_0.DriveHalt := FALSE;
                    // _AxisReference^.Outputs.DriveControlWord_S_0_0134_0_0.DriveEnable := FALSE;
                    // _AxisReference^.Outputs.DriveControlWord_S_0_0134_0_0.DriveOn := FALSE;
                    _AxisReference^.Outputs.SignalControlWord_S_0_0145_0_0.AcceptanceOfPositioningCommandValue := FALSE;
                    _AxisReference^.Outputs.SignalControlWord_S_0_0145_0_0.HomingControl := FALSE;
                    _AxisReference^.Outputs.SignalControlWord_S_0_0145_0_0.AbsoluteRelative := FALSE;
                    _AxisReference^.Outputs.SignalControlWord_S_0_0145_0_0.ImmediateChange := FALSE;
                    _AxisReference^.Outputs.SignalControlWord_S_0_0145_0_0.JogPositive := FALSE;
                    _AxisReference^.Outputs.SignalControlWord_S_0_0145_0_0.JogNegative := FALSE;
                    _AxisReference^.Outputs.SignalControlWord_S_0_0145_0_0.ClearError := FALSE;
                    _State := UINT#310;
                    THIS.CallTimers(FALSE);
                END_IF;
                // Reseting InReference flag
                IF _State = UINT#310 THEN
                    IF _infoTimer.output THEN
                        TaskMessenger.Activate( UINT#510, eAxoMessageCategory#Potential);
                        DriveStatus.Error.Id := UINT#510;
                    END_IF;
                    _AxisReference^.Outputs.SignalControlWord_S_0_0145_0_0.CancelReferencePoint := TRUE;
                    IF NOT _AxisReference^.Inputs.DriveStatusWord_S_0_0135_0_0.InReference THEN
                        _AxisReference^.Outputs.SignalControlWord_S_0_0145_0_0.CancelReferencePoint := FALSE;
                        _State := UINT#311;
                        THIS.CallTimers(FALSE);
                        RETURN;
                    END_IF;
                END_IF;
                //Writing Homing configuration ENC_1: Home offset (0x607C:00 / S-0-0052 / --)
                IF _State = UINT#311 THEN
                    IF _infoTimer.output THEN
                        TaskMessenger.Activate( UINT#511, eAxoMessageCategory#Potential);
                        DriveStatus.Error.Id := UINT#511;
                    END_IF;
                    IF Acceleration <= 0 OR Deceleration <= 0 THEN
                        _State := UINT#329;
                        THIS.CallTimers(FALSE);
                        RETURN;
                    END_IF;

                    _dword :=  TO_DWORD(TO_DINT(Position * ScalingConstantRequiredPosition));
                    _data4[0] := _dword.%B0;
                    _data4[1] := _dword.%B1;
                    _data4[2] := _dword.%B2;
                    _data4[3] := _dword.%B3;
                    _WriteRecord(   request     :=  TRUE,
                                    hardwareID  :=  (AxisRefExt.HWIDs.HW_S_0_0134_0_0),
                                    index       :=  DINT#52,
                                    length      :=  UINT#4,
                                    record      :=  _data4);
                    IF NOT _WriteRecord.busy AND _WriteRecord.done AND NOT _WriteRecord.error THEN
                        _State := UINT#312;
                        THIS.CallTimers(FALSE);
                    ElSIF _WriteRecord.error THEN
                        Messenger.Activate( UINT#1444, eAxoMessageCategory#Error);
                        MC_HomeErrorID :=   DINT#1444;
                        _WriteRecord(request := FALSE, record := _data4);
                        _State := UINT#329;
                        THIS.CallTimers(FALSE);
                    END_IF;
                END_IF;
                IF _State = UINT#312 THEN
                    IF _infoTimer.output THEN
                        TaskMessenger.Activate( UINT#512, eAxoMessageCategory#Potential);
                        DriveStatus.Error.Id := UINT#512;
                    END_IF;
                    _WriteRecord(request := FALSE, record := _data4);
                    IF NOT _WriteRecord.busy AND NOT _WriteRecord.done AND NOT _WriteRecord.error  THEN
                        _State := UINT#313;
                        THIS.CallTimers(FALSE);
                    END_IF;
                END_IF;
                //Writing Homing function: Configuration (0x2500:02 / S-0-0147 / --)
                IF _State = UINT#313 THEN
                    IF _infoTimer.output THEN
                        TaskMessenger.Activate( UINT#513, eAxoMessageCategory#Potential);
                        DriveStatus.Error.Id := UINT#513;
                    END_IF;
                    _word :=  TO_WORD(HommingMode);
                    _data2[0] := _word.%B0;
                    _data2[1] := _word.%B1;
                    _WriteRecord(   request     :=  TRUE,
                                    hardwareID  :=  (AxisRefExt.HWIDs.HW_S_0_0134_0_0),
                                    index       :=  DINT#147,
                                    length      :=  UINT#2,
                                    record      :=  _data2);
                    IF NOT _WriteRecord.busy AND _WriteRecord.done AND NOT _WriteRecord.error THEN
                        _State := UINT#314;
                        THIS.CallTimers(FALSE);
                    ElSIF _WriteRecord.error THEN
                        Messenger.Activate( UINT#1445, eAxoMessageCategory#Error);
                        MC_HomeErrorID :=   DINT#1445;
                        _WriteRecord(request := FALSE, record := _data2);
                        _State := UINT#329;
                        THIS.CallTimers(FALSE);
                    END_IF;
                END_IF;
                IF _State = UINT#314 THEN
                    IF _infoTimer.output THEN
                        TaskMessenger.Activate( UINT#514, eAxoMessageCategory#Potential);
                        DriveStatus.Error.Id := UINT#514;
                    END_IF;
                    _WriteRecord(request := FALSE, record := _data2);
                    IF NOT _WriteRecord.busy AND NOT _WriteRecord.done AND NOT _WriteRecord.error  THEN
                        _State := UINT#315;
                        THIS.CallTimers(FALSE);
                    END_IF;
                END_IF;
                //Writing Homing speeds: Speed during search for switch (0x6099:01 / S-0-0041 / --)
                IF _State = UINT#315 THEN
                    IF _infoTimer.output THEN
                        TaskMessenger.Activate( UINT#515, eAxoMessageCategory#Potential);
                        DriveStatus.Error.Id := UINT#515;
                    END_IF;
                    _dword :=  TO_DWORD(TO_DINT(Velocity * ScalingConstantRequiredVelocity));
                    _data4[0] := _dword.%B0;
                    _data4[1] := _dword.%B1;
                    _data4[2] := _dword.%B2;
                    _data4[3] := _dword.%B3;
                    _WriteRecord(   request     :=  TRUE,
                                    hardwareID  :=  (AxisRefExt.HWIDs.HW_S_0_0134_0_0),
                                    index       :=  DINT#41,
                                    length      :=  UINT#4,
                                    record      :=  _data4);
                    IF NOT _WriteRecord.busy AND _WriteRecord.done AND NOT _WriteRecord.error THEN
                        _WriteRecord(request := FALSE, record := _data4);
                        _State := UINT#316;
                        THIS.CallTimers(FALSE);
                    ElSIF _WriteRecord.error THEN
                        Messenger.Activate( UINT#1446, eAxoMessageCategory#Error);
                        MC_HomeErrorID :=   DINT#1446;
                        _WriteRecord(request := FALSE, record := _data4);
                        _State := UINT#329;
                        THIS.CallTimers(FALSE);
                    END_IF;
                END_IF;
                //Writing Homing speeds: Speed during search for zero (0x6099:02 / S-0-0542 / --)
                IF _State = UINT#316 THEN
                    IF _infoTimer.output THEN
                        TaskMessenger.Activate( UINT#516, eAxoMessageCategory#Potential);
                        DriveStatus.Error.Id := UINT#516;
                    END_IF;
                    _dword :=  TO_DWORD(TO_DINT(Velocity * ScalingConstantRequiredVelocity * 0.1));
                    _data4[0] := _dword.%B0;
                    _data4[1] := _dword.%B1;
                    _data4[2] := _dword.%B2;
                    _data4[3] := _dword.%B3;
                    _WriteRecord(   request     :=  TRUE,
                                    hardwareID  :=  (AxisRefExt.HWIDs.HW_S_0_0134_0_0),
                                    index       :=  DINT#542,
                                    length      :=  UINT#4,
                                    record      :=  _data4);
                    IF NOT _WriteRecord.busy AND _WriteRecord.done AND NOT _WriteRecord.error THEN
                        _WriteRecord(request := FALSE, record := _data4);
                        _State := UINT#317;
                        THIS.CallTimers(FALSE);
                    ElSIF _WriteRecord.error THEN
                        Messenger.Activate( UINT#1446, eAxoMessageCategory#Error);
                        MC_HomeErrorID :=   DINT#1446;
                        _WriteRecord(request := FALSE, record := _data4);
                        _State := UINT#329;
                        THIS.CallTimers(FALSE);
                    END_IF;
                END_IF;
                //Writing Homing acceleration (0x609A:00 / S-0-0042 / --)
                IF _State = UINT#317 THEN
                    IF _infoTimer.output THEN
                        TaskMessenger.Activate( UINT#517, eAxoMessageCategory#Potential);
                        DriveStatus.Error.Id := UINT#517;
                    END_IF;
                    _dword :=  TO_DWORD(TO_DINT(Acceleration * ScalingConstantRequiredAcceleration));
                    _data4[0] := _dword.%B0;
                    _data4[1] := _dword.%B1;
                    _data4[2] := _dword.%B2;
                    _data4[3] := _dword.%B3;
                    _WriteRecord(   request     :=  TRUE,
                                    hardwareID  :=  (AxisRefExt.HWIDs.HW_S_0_0134_0_0),
                                    index       :=  DINT#42,
                                    length      :=  UINT#4,
                                    record      :=  _data4);
                    IF NOT _WriteRecord.busy AND _WriteRecord.done AND NOT _WriteRecord.error THEN
                        _State := UINT#318;
                        THIS.CallTimers(FALSE);
                    ElSIF _WriteRecord.error THEN
                        Messenger.Activate( UINT#1447, eAxoMessageCategory#Error);
                        MC_HomeErrorID :=   DINT#1447;
                        _WriteRecord(request := FALSE, record := _data4);
                        _State := UINT#329;
                        THIS.CallTimers(FALSE);
                    END_IF;
                END_IF;
                IF _State = UINT#318 THEN
                    IF _infoTimer.output THEN
                        TaskMessenger.Activate( UINT#518, eAxoMessageCategory#Potential);
                        DriveStatus.Error.Id := UINT#518;
                    END_IF;
                    _WriteRecord(request := FALSE, record := _data4);
                    IF NOT _WriteRecord.busy AND NOT _WriteRecord.done AND NOT _WriteRecord.error  THEN
                        _State := UINT#319;
                        THIS.CallTimers(FALSE);
                    END_IF;
                END_IF;
                IF _State = UINT#319 THEN
                    IF _infoTimer.output THEN
                        TaskMessenger.Activate( UINT#519, eAxoMessageCategory#Potential);
                        DriveStatus.Error.Id := UINT#519;
                    END_IF;
                    _AxisReference^.Outputs.DriveControlWord_S_0_0134_0_0.CommandOperationModeBit0  := FALSE;
                    _AxisReference^.Outputs.DriveControlWord_S_0_0134_0_0.CommandOperationModeBit1  := FALSE;
                    _AxisReference^.Outputs.DriveControlWord_S_0_0134_0_0.CommandOperationModeBit2  := FALSE;
                    IF  NOT _AxisReference^.Inputs.DriveStatusWord_S_0_0135_0_0.ActualOperatingModeBit0 AND
                        NOT _AxisReference^.Inputs.DriveStatusWord_S_0_0135_0_0.ActualOperatingModeBit1 AND
                        NOT _AxisReference^.Inputs.DriveStatusWord_S_0_0135_0_0.ActualOperatingModeBit2 THEN
                        _State := UINT#320;
                        THIS.CallTimers(FALSE);
                    END_IF;
                END_IF;
                IF _State = UINT#320 THEN
                    IF _infoTimer.output THEN
                        TaskMessenger.Activate( UINT#520, eAxoMessageCategory#Potential);
                        DriveStatus.Error.Id := UINT#520;
                    END_IF;
                    IF  _AxisReference^.Inputs.DriveStatusWord_S_0_0135_0_0.ReadyForOperationBit0 AND
                        _AxisReference^.Inputs.DriveStatusWord_S_0_0135_0_0.ReadyForOperationBit1 THEN
                       _State := UINT#321;
                        THIS.CallTimers(FALSE);
                    END_IF;
                END_IF;
                IF _State = UINT#321 THEN
                    IF _infoTimer.output THEN
                        TaskMessenger.Activate( UINT#521, eAxoMessageCategory#Potential);
                        DriveStatus.Error.Id := UINT#521;
                    END_IF;
                    _AxisReference^.Outputs.DriveControlWord_S_0_0134_0_0.DriveHalt  := TRUE;
                    IF _AxisReference^.Inputs.DriveStatusWord_S_0_0135_0_0.CommandProcessingStatus AND NOT _AxisReference^.Inputs.DriveStatusWord_S_0_0135_0_0.InStandstill  THEN
                       _State := UINT#322;
                        THIS.CallTimers(FALSE);
                    END_IF;
                END_IF;
                IF _State = UINT#322 THEN
                    IF _infoTimer.output THEN
                        TaskMessenger.Activate( UINT#522, eAxoMessageCategory#Potential);
                        DriveStatus.Error.Id := UINT#522;
                    END_IF;
                    _AxisReference^.Outputs.SignalControlWord_S_0_0145_0_0.HomingControl := TRUE;
                    _AxisReference^.Outputs.SignalControlWord_S_0_0145_0_0.AcceptanceOfPositioningCommandValue := NOT _AxisReference^.Outputs.SignalControlWord_S_0_0145_0_0.AcceptanceOfPositioningCommandValue;
                   _State := UINT#323;
                    THIS.CallTimers(FALSE);
                END_IF;
                IF _State = UINT#323 THEN
                    IF _infoTimer.output THEN
                        TaskMessenger.Activate( UINT#523, eAxoMessageCategory#Potential);
                        DriveStatus.Error.Id := UINT#523;
                    END_IF;
                    IF _AxisReference^.Inputs.DriveStatusWord_S_0_0135_0_0.InReference AND _AxisReference^.Inputs.SignalStatusWord_S_0_0144_0_0.DriveStandstill THEN
                        _AxisReference^.Outputs.SignalControlWord_S_0_0145_0_0.HomingControl := FALSE;
                        _State := UINT#324;
                        THIS.CallTimers(FALSE);
                    END_IF;
                END_IF;
                IF _State = UINT#324 THEN
                    _AxisReference^.Outputs.SignalControlWord_S_0_0145_0_0.AcceptanceOfPositioningCommandValue := FALSE;
                    _AxisReference^.Outputs.SignalControlWord_S_0_0145_0_0.HomingControl := FALSE;
                    _AxisReference^.Outputs.SignalControlWord_S_0_0145_0_0.AbsoluteRelative := FALSE;
                    _AxisReference^.Outputs.SignalControlWord_S_0_0145_0_0.ImmediateChange := FALSE;
                    _AxisReference^.Outputs.SignalControlWord_S_0_0145_0_0.JogPositive := FALSE;
                    _AxisReference^.Outputs.SignalControlWord_S_0_0145_0_0.JogNegative := FALSE;
                    _AxisReference^.Outputs.SignalControlWord_S_0_0145_0_0.ClearError := FALSE;
                    _State := UINT#325;
                    THIS.CallTimers(FALSE);
                END_IF;
                IF _State = UINT#325 THEN
                    _tmpTimer.OnDelay(THIS,  _AxisReference^.Inputs.DriveStatusWord_S_0_0135_0_0.InReference AND _AxisReference^.Inputs.SignalStatusWord_S_0_0144_0_0.DriveStandstill , T#100ms);
                    IF _tmpTimer.output THEN
                        _State := UINT#326;
                        THIS.CallTimers(FALSE);
                    END_IF;
                END_IF;
                IF _State = UINT#326 THEN
                    _State := UINT#327;
                    THIS.CallTimers(FALSE);
                END_IF;
                IF _State = UINT#327 THEN
                    Done := TRUE;
                    MC_HomeCycle := ULINT#0;
                END_IF;
                IF _State = UINT#328 THEN
                    _AxisReference^.Outputs.SignalControlWord_S_0_0145_0_0.HomingControl := FALSE;
                    MC_HomeCycle := ULINT#0;
                    CommandAborted := TRUE; // action handled in parent AxoDrive
                END_IF;
                IF _State = UINT#329 THEN
                    _AxisReference^.Outputs.SignalControlWord_S_0_0145_0_0.HomingControl := FALSE;
                    MC_HomeCycle := ULINT#0;
                    Error := TRUE; // action handled in parent AxoDrive
                END_IF;

                IF _State>=UINT#310 AND _State<UINT#327 THEN
                    IF NOT _AxisReference^.Inputs.DriveStatusWord_S_0_0135_0_0.ReadyForOperationBit0 OR NOT _AxisReference^.Inputs.DriveStatusWord_S_0_0135_0_0.ReadyForOperationBit1 THEN
                        _State := UINT#328;
                    ELSIF _AxisReference^.Inputs.DriveStatusWord_S_0_0135_0_0.DriveErrorZKL1 OR
                        (_AxisReference^.Inputs.DriveStatusWord_S_0_0135_0_0.WarningZKL2 AND _AxisReference^.Inputs.DiagnosticMessage_S_0_0390_0_0 >= DWORD#16#C00E0000)
                        // Filtering out warning with code C00E2054 (NOT HOMED)
                        AND (_AxisReference^.Inputs.DiagnosticMessage_S_0_0390_0_0 <> DWORD#16#C00E2054) THEN
                        IF MC_HomeErrorID = DINT#0 THEN
                            MC_HomeErrorID := TO_DINT(_AxisReference^.Inputs.DiagnosticMessage_S_0_0390_0_0 AND DWORD#16#000FFFFF);
                        END_IF;
                        _State := UINT#329;
                    ELSIF _AxisReference^.Data.Cycle <> MC_HomeCycle THEN
                        _AxisReference^.Data.Cycle := _AxisReference^.Data.Cycle - ULINT#1;
                        _State := UINT#328;
                    END_IF;
                END_IF;

                THIS.CallTimers(TRUE,FALSE);
                THIS.AxoHome_Task.ThrowWhen(_errorTimer.output );
                // THIS.AxoHome_Task.ThrowWhen(THIS.AxoHome_Task.Duration >= DriveConfig.TaskTimeout AND DriveConfig.TaskTimeout > T#0s ,'<#AxoHome_Task timeout.#>');
                DriveStatus.Action.Id := _State;
            END_IF;

            IF THIS.AxoHome_Task.DoneReached() AND _State>=UINT#310 AND _State<=UINT#329 THEN
                _AxisReference^.Status.CurrentMotionTaskId := AXOpen.Components.Drives.eAxoMotionTaskId#Axo_Done;
                _AxisReference^.Outputs.SignalControlWord_S_0_0145_0_0.HomingControl := FALSE;
                _AxisReference^.Outputs.SignalControlWord_S_0_0145_0_0.CancelReferencePoint := FALSE;
                MC_HomeErrorID := DINT#0;
                _State := UINT#0;
            END_IF;
            IF THIS.AxoHome_Task.RestoreTriggered() AND _State>=UINT#310 AND _State<=UINT#329 THEN
                _AxisReference^.Status.CurrentMotionTaskId := AXOpen.Components.Drives.eAxoMotionTaskId#Axo_None;
                _AxisReference^.Outputs.SignalControlWord_S_0_0145_0_0.HomingControl := FALSE;
                _AxisReference^.Outputs.SignalControlWord_S_0_0145_0_0.CancelReferencePoint := FALSE;
                MC_HomeErrorID := DINT#0;
                _State := UINT#0;
                MC_HomeCycle := ULINT#0;
            END_IF;

            ErrorID := MC_HomeErrorID;
            MC_HomeExecute_PV := Execute;
        END_METHOD

        ///<summary>
        /// This method commands a controlled motion stop and transfers the axis to the State ‘Stopping’. It aborts any
        /// ongoing method execution. While the axis is in State ‘Stopping’, no other method can perform any motion on the
        /// same axis.
        ///</summary>
        VAR INTERNAL
            MC_StopExecute_PV					: 	BOOL;				//Execute - previous value
            MC_StopErrorID					    : 	DINT;
            MC_StopCycle					    : 	ULINT;
        END_VAR
        METHOD PUBLIC OVERRIDE MC_Stop
            VAR_INPUT
                AxisRef         :   AXOpen.Components.Abstractions.Drives.IAxoAxisReference;
                Execute         :   BOOL;                       //  Start the action at rising edge
                Deceleration    :   LREAL;                      //  Value of the ‘Deceleration’ [u/s2]
                Jerk            :   LREAL;                      //  Value of the ‘Jerk’ [u/s3]
            END_VAR
            VAR_OUTPUT
                Done            :   BOOL;                       // Zero velocity reached
                Busy            :   BOOL;                       // The method is not finished and new output values are to be expected
                Active          :   BOOL;                       // Indicates that the method has control on the axis
                CommandAborted  :   BOOL;                       // ‘Command’ is aborted by switching off power (only possibility to abort)
                Error           :   BOOL;                       // Signals that an error has occurred within the method
                ErrorID         :   DINT;                       // Error identification
            END_VAR
            VAR
                _AxisReference :  REF_TO AxoCtrlxDriveXscAxisReference;
            END_VAR

            _AxisReference ?= AxisRef;

            IF(_AxisReference = NULL) THEN
                Messenger.Activate(     UINT#1470, eAxoMessageCategory#ProgrammingError);
                DriveStatus.Error.Id := UINT#1470;
                RETURN;
            END_IF;

            IF THIS.AxoStop_Task.StartTriggered() THEN
                _AxisReference^.Status.CurrentMotionTaskId := AXOpen.Components.Drives.eAxoMotionTaskId#Axo_Stop;
            END_IF;

            IF Execute AND NOT MC_StopExecute_PV THEN
                _AxisReference^.Data.Cycle := _AxisReference^.Data.Cycle + ULINT#2;
                MC_StopCycle := _AxisReference^.Data.Cycle ;
                _State := UINT#0;
            END_IF;

            IF Execute THEN
                Messenger.ActivateOnCondition(ULINT#1471, Execute AND Deceleration <= 0, eAxoMessageCategory#ProgrammingError);
                Messenger.ActivateOnCondition(ULINT#1472, Execute AND Jerk <= 0, eAxoMessageCategory#ProgrammingError);

                IF _State = UINT#0 THEN
                    Busy := TRUE;
                    Active := TRUE;
                    MC_StopErrorID := DINT#0;
                    _AxisReference^.Outputs.SignalControlWord_S_0_0145_0_0.HomingControl := FALSE;
                    _AxisReference^.Outputs.SignalControlWord_S_0_0145_0_0.JogPositive := FALSE;
                    _AxisReference^.Outputs.SignalControlWord_S_0_0145_0_0.JogNegative := FALSE;
                    _AxisReference^.Outputs.CommandDecceleration_S_0_0359_0_0 := TO_DINT(Deceleration * ScalingConstantRequiredDeceleration );
                    _AxisReference^.Outputs.CommandJerk_S_0_0193_0_0 := TO_DINT(Jerk * ScalingConstantRequiredJerk );
                    _State := UINT#330;
                    THIS.CallTimers(FALSE);
                END_IF;
                IF _State = UINT#330 THEN
                    Busy := TRUE;
                    Active := TRUE;
                    IF Deceleration <= 0 OR Jerk <= 0 THEN
                        _State := UINT#339;
                        THIS.CallTimers(FALSE);
                    ELSE
                        _State := UINT#331;
                        THIS.CallTimers(FALSE);
                    END_IF;
                END_IF;
                IF _State = UINT#331 THEN
                    IF _infoTimer.output THEN
                        TaskMessenger.Activate( UINT#531, eAxoMessageCategory#Potential);
                        DriveStatus.Error.Id := UINT#531;
                    END_IF;
                    Busy := TRUE;
                    Active := TRUE;
                    _AxisReference^.Outputs.DriveControlWord_S_0_0134_0_0.DriveHalt := FALSE;
                    IF _AxisReference^.Inputs.DriveStatusWord_S_0_0135_0_0.InStandstill THEN
                        _State := UINT#332;
                        THIS.CallTimers(FALSE);
                    END_IF;
                END_IF;
                IF _State = UINT#332 THEN
                    Busy := TRUE;
                    Active := TRUE;
                    IF TRUE THEN
                        _State := UINT#333;
                        THIS.CallTimers(FALSE);
                    END_IF;
                END_IF;
                IF _State = UINT#333 THEN
                    Busy := TRUE;
                    Active := TRUE;
                    IF TRUE THEN
                        _State := UINT#334;
                        THIS.CallTimers(FALSE);
                    END_IF;
                END_IF;
                IF _State = UINT#334 THEN
                    Busy := TRUE;
                    Active := TRUE;
                    IF TRUE THEN
                        _State := UINT#335;
                        THIS.CallTimers(FALSE);
                    END_IF;
                END_IF;
                IF _State = UINT#335 THEN
                    Busy := TRUE;
                    Active := TRUE;
                    IF TRUE THEN
                        _State := UINT#336;
                        THIS.CallTimers(FALSE);
                    END_IF;
                END_IF;
                IF _State = UINT#336 THEN
                    Busy := TRUE;
                    Active := TRUE;
                    IF TRUE THEN
                        _State := UINT#337;
                        THIS.CallTimers(FALSE);
                    END_IF;
                END_IF;
                IF _State = UINT#337 THEN
                    Done := TRUE;
                    Active := TRUE;
                    MC_StopCycle := ULINT#0;
                    THIS.CallTimers(FALSE);
                END_IF;
                IF _State = UINT#338 THEN
                    MC_StopCycle := ULINT#0;
                    CommandAborted := TRUE; // action handled in parent AxoDrive
                END_IF;
                IF _State = UINT#339 THEN
                    MC_StopCycle := ULINT#0;
                    Error := TRUE; // action handled in parent AxoDrive
                END_IF;

                IF _State>=UINT#330 AND _State<UINT#337 THEN
                    IF NOT _AxisReference^.Inputs.DriveStatusWord_S_0_0135_0_0.ReadyForOperationBit0 OR NOT _AxisReference^.Inputs.DriveStatusWord_S_0_0135_0_0.ReadyForOperationBit1 THEN
                        _State := UINT#338;
                    ELSIF _AxisReference^.Inputs.DriveStatusWord_S_0_0135_0_0.DriveErrorZKL1 OR
                        (_AxisReference^.Inputs.DriveStatusWord_S_0_0135_0_0.WarningZKL2 AND _AxisReference^.Inputs.DiagnosticMessage_S_0_0390_0_0 >= DWORD#16#C00E0000) THEN
                        IF MC_StopErrorID = DINT#0 THEN
                            MC_StopErrorID := TO_DINT(_AxisReference^.Inputs.DiagnosticMessage_S_0_0390_0_0 AND DWORD#16#000FFFFF);
                        END_IF;
                        _State := UINT#339;
                    ELSIF _AxisReference^.Data.Cycle <> MC_StopCycle THEN
                        _AxisReference^.Data.Cycle := _AxisReference^.Data.Cycle - ULINT#1;
                        _State := UINT#338;
                    END_IF;
                END_IF;
                THIS.CallTimers(TRUE,FALSE);
                THIS.AxoStop_Task.ThrowWhen(_errorTimer.output );
                THIS.AxoStop_Task.ThrowWhen(THIS.AxoStop_Task.Duration >= DriveConfig.TaskTimeout AND DriveConfig.TaskTimeout > T#0s ,'<#AxoStop_Task timeout.#>');
                DriveStatus.Action.Id := _State;
            END_IF;

            IF THIS.AxoStop_Task.DoneReached() AND _State>=UINT#330 AND _State<=UINT#339 THEN
                _AxisReference^.Status.CurrentMotionTaskId := AXOpen.Components.Drives.eAxoMotionTaskId#Axo_Done;
                MC_StopErrorID := DINT#0;
                _State := UINT#0;
            END_IF;
            IF THIS.AxoStop_Task.RestoreTriggered() AND _State>=UINT#330 AND _State<=UINT#339 THEN
                _AxisReference^.Status.CurrentMotionTaskId := AXOpen.Components.Drives.eAxoMotionTaskId#Axo_None;
                MC_StopErrorID := DINT#0;
                _State := UINT#0;
                MC_StopCycle := ULINT#0;
            END_IF;
            ErrorID := MC_StopErrorID;
            MC_StopExecute_PV := Execute;
        END_METHOD

        ///<summary>
        /// This method commands a controlled motion stop. The axis is moved to the State ‘DiscreteMotion’, until the
        /// velocity is zero. With the ‘Done’ output set, the State is transferred to ‘Standstill’.
        ///</summary>
        VAR INTERNAL
            MC_HaltExecute_PV					: 	BOOL;				//Execute - previous value
            MC_HaltErrorID					    : 	DINT;
            MC_HaltCycle					    : 	ULINT;
        END_VAR
        METHOD PUBLIC OVERRIDE MC_Halt
            VAR_INPUT
                AxisRef         :   AXOpen.Components.Abstractions.Drives.IAxoAxisReference;
                Execute         :   BOOL;                       //  Start the action at rising edge
                Deceleration    :   LREAL;                      //  Value of the ‘Deceleration’ [u/s2]
                Jerk            :   LREAL;                      //  Value of the ‘Jerk’ [u/s3]
            END_VAR
            VAR_OUTPUT
                Done            :   BOOL;                       // Zero velocity reached
                Busy            :   BOOL;                       // The method is not finished and new output values are to be expected
                Active          :   BOOL;                       // Indicates that the method has control on the axis
                CommandAborted  :   BOOL;                       // ‘Command’ is aborted by switching off power (only possibility to abort)
                Error           :   BOOL;                       // Signals that an error has occurred within the method
                ErrorID         :   DINT;                       // Error identification
            END_VAR
            VAR
                _AxisReference :  REF_TO AxoCtrlxDriveXscAxisReference;
            END_VAR

            _AxisReference ?= AxisRef;

            IF(_AxisReference = NULL) THEN
                Messenger.Activate(     UINT#1480, eAxoMessageCategory#ProgrammingError);
                DriveStatus.Error.Id := UINT#1480;
                RETURN;
            END_IF;

            IF THIS.AxoHalt_Task.StartTriggered() THEN
                _AxisReference^.Status.CurrentMotionTaskId := AXOpen.Components.Drives.eAxoMotionTaskId#Axo_Halt;
            END_IF;

            IF Execute AND NOT MC_HaltExecute_PV THEN
                _AxisReference^.Data.Cycle := _AxisReference^.Data.Cycle + ULINT#2;
                MC_HaltCycle := _AxisReference^.Data.Cycle ;
                _State := UINT#0;
            END_IF;

            IF Execute THEN
                Messenger.ActivateOnCondition(ULINT#1481, Execute AND Deceleration <= 0, eAxoMessageCategory#ProgrammingError);
                Messenger.ActivateOnCondition(ULINT#1482, Execute AND Jerk <= 0, eAxoMessageCategory#ProgrammingError);

                IF _State = UINT#0 THEN
                    Busy := TRUE;
                    Active := TRUE;
                    MC_HaltErrorID := DINT#10;
                    _AxisReference^.Outputs.SignalControlWord_S_0_0145_0_0.HomingControl := FALSE;
                    _AxisReference^.Outputs.SignalControlWord_S_0_0145_0_0.JogPositive := FALSE;
                    _AxisReference^.Outputs.SignalControlWord_S_0_0145_0_0.JogNegative := FALSE;
                    _AxisReference^.Outputs.CommandDecceleration_S_0_0359_0_0 := TO_DINT(Deceleration * ScalingConstantRequiredDeceleration);
                    _AxisReference^.Outputs.CommandJerk_S_0_0193_0_0 := TO_DINT(Jerk * ScalingConstantRequiredJerk);
                    _State := UINT#340;
                    THIS.CallTimers(FALSE);
                END_IF;
                IF _State = UINT#340 THEN
                    IF _infoTimer.output THEN
                        TaskMessenger.Activate( UINT#540, eAxoMessageCategory#Potential);
                        DriveStatus.Error.Id := UINT#540;
                    END_IF;
                    Busy := TRUE;
                    Active := TRUE;
                    IF Deceleration <= 0 OR Jerk <= 0 THEN
                        _State := UINT#349;
                        THIS.CallTimers(FALSE);
                    ELSE
                        _State := UINT#341;
                        THIS.CallTimers(FALSE);
                    END_IF;
                END_IF;
                IF _State = UINT#341 THEN
                    IF _infoTimer.output THEN
                        TaskMessenger.Activate( UINT#541, eAxoMessageCategory#Potential);
                        DriveStatus.Error.Id := UINT#541;
                    END_IF;
                    Busy := TRUE;
                    Active := TRUE;
                    _AxisReference^.Outputs.DriveControlWord_S_0_0134_0_0.DriveHalt := FALSE;
                    IF _AxisReference^.Inputs.DriveStatusWord_S_0_0135_0_0.InStandstill THEN
                        _State := UINT#342;
                        THIS.CallTimers(FALSE);
                    END_IF;
                END_IF;
                IF _State = UINT#342 THEN
                    Busy := TRUE;
                    Active := TRUE;
                    IF TRUE THEN
                        _State := UINT#343;
                        THIS.CallTimers(FALSE);
                    END_IF;
                END_IF;
                IF _State = UINT#343 THEN
                    Busy := TRUE;
                    Active := TRUE;
                    IF TRUE THEN
                        _State := UINT#344;
                        THIS.CallTimers(FALSE);
                    END_IF;
                END_IF;
                IF _State = UINT#344 THEN
                    IF TRUE THEN
                        _State := UINT#345;
                        THIS.CallTimers(FALSE);
                    END_IF;
                END_IF;
                IF _State = UINT#345 THEN
                    IF TRUE THEN
                        _State := UINT#346;
                        THIS.CallTimers(FALSE);
                    END_IF;
                END_IF;
                IF _State = UINT#346 THEN
                    IF TRUE THEN
                        _State := UINT#347;
                        THIS.CallTimers(FALSE);
                    END_IF;
                END_IF;
                IF _State = UINT#347 THEN
                    Done := TRUE;
                    _AxisReference^.Outputs.DriveControlWord_S_0_0134_0_0.DriveHalt := TRUE;
                    MC_HaltCycle := ULINT#0;
                END_IF;
                IF _State = UINT#348 THEN
                    _AxisReference^.Outputs.DriveControlWord_S_0_0134_0_0.DriveHalt := TRUE;
                    CommandAborted := TRUE;
                    THIS.AxoHalt_Task.Abort();
                END_IF;
                IF _State = UINT#349 THEN
                    _AxisReference^.Outputs.DriveControlWord_S_0_0134_0_0.DriveHalt := TRUE;
                    MC_HaltCycle := ULINT#0;
                    Error := TRUE;
                    THIS.AxoHalt_Task.ThrowWhen(TRUE);
                END_IF;
                IF _State>=UINT#340 AND _State<UINT#347 THEN
                    IF NOT _AxisReference^.Inputs.DriveStatusWord_S_0_0135_0_0.ReadyForOperationBit0 OR NOT _AxisReference^.Inputs.DriveStatusWord_S_0_0135_0_0.ReadyForOperationBit1 THEN
                        _State := UINT#348;
                    ELSIF _AxisReference^.Inputs.DriveStatusWord_S_0_0135_0_0.DriveErrorZKL1 OR
                        (_AxisReference^.Inputs.DriveStatusWord_S_0_0135_0_0.WarningZKL2 AND _AxisReference^.Inputs.DiagnosticMessage_S_0_0390_0_0 >= DWORD#16#C00E0000) THEN
                        IF MC_HaltErrorID = DINT#0 THEN
                            MC_HaltErrorID := TO_DINT(_AxisReference^.Inputs.DiagnosticMessage_S_0_0390_0_0 AND DWORD#16#000FFFFF);
                        END_IF;
                        _State := UINT#349;
                    ELSIF _AxisReference^.Data.Cycle <> MC_HaltCycle THEN
                        _AxisReference^.Data.Cycle := _AxisReference^.Data.Cycle - ULINT#1;
                        _State := UINT#348;
                    END_IF;
                END_IF;
                THIS.CallTimers(TRUE,FALSE);
                THIS.AxoHalt_Task.ThrowWhen(_errorTimer.output );
                THIS.AxoHalt_Task.ThrowWhen(THIS.AxoHalt_Task.Duration >= DriveConfig.TaskTimeout AND DriveConfig.TaskTimeout > T#0s ,'<#AxoHalt_Task timeout.#>');
                DriveStatus.Action.Id := _State;
            END_IF;

            IF THIS.AxoHalt_Task.DoneReached() AND _State>=UINT#340 AND _State<=UINT#349 THEN
                _AxisReference^.Status.CurrentMotionTaskId := AXOpen.Components.Drives.eAxoMotionTaskId#Axo_Done;
                _AxisReference^.Outputs.DriveControlWord_S_0_0134_0_0.DriveHalt := TRUE;
                MC_HaltErrorID := DINT#0;
                _State := UINT#0;
            END_IF;
            IF THIS.AxoHalt_Task.RestoreTriggered() AND _State>=UINT#340 AND _State<=UINT#349 THEN
                _AxisReference^.Status.CurrentMotionTaskId := AXOpen.Components.Drives.eAxoMotionTaskId#Axo_None;
                _AxisReference^.Outputs.DriveControlWord_S_0_0134_0_0.DriveHalt := TRUE;
                MC_HaltErrorID := DINT#0;
                _State := UINT#0;
                MC_HaltCycle := ULINT#0;
            END_IF;
            ErrorID := MC_HaltErrorID;
            MC_HaltExecute_PV := Execute;
        END_METHOD

        ///<summary>
        /// This method commands a controlled motion to a specified absolute position.
        ///</summary>
        VAR INTERNAL
            MC_MoveAbsoluteExecute_PV					: 	BOOL;				//Execute - previous value
            MC_MoveAbsoluteErrorID					    : 	DINT;
            MC_MoveAbsoluteCycle					    : 	ULINT;
            MC_MoveAbsoluteContinuousUpdate_SV          :   BOOL;
            MC_MoveAbsolutePosition_PV                  :   LREAL;
            MC_MoveAbsoluteVelocity_PV                  :   LREAL;
            MC_MoveAbsoluteAcceleration_PV              :   LREAL;
            MC_MoveAbsoluteDeceleration_PV              :   LREAL;
            MC_MoveAbsoluteJerk_PV                      :   LREAL;
            MC_MoveAbsoluteDirection_PV                 :   AXOpen.Components.Abstractions.Drives.eAxoDriveDirection;
        END_VAR
        METHOD PUBLIC OVERRIDE MC_MoveAbsolute
            VAR_INPUT
                AxisRef         :   AXOpen.Components.Abstractions.Drives.IAxoAxisReference;
                Execute         :   BOOL;                       //  Start the motion at rising edge
                ContinuousUpdate:   BOOL;                       //  Activate ‘ContinuousUpdate’ - target parameters should be changed during movement
                Position        :   LREAL;                      //  Commanded ‘Position’ for the motion (in technical unit [u]) (negative or positive)
                Velocity        :   LREAL;                      //  Value of the maximum ‘Velocity’ (not necessarily reached) [u/s].
                Acceleration    :   LREAL;                      //  Value of the ‘Acceleration’ (always positive) (increasing energy of the motor) [u/s2]
                Deceleration    :   LREAL;                      //  Value of the ‘Deceleration’ (always positive) (decreasing energy of the motor) [u/s2]
                Jerk            :   LREAL;                      //  Value of the ‘Jerk’ [u/s3]
                Direction       :   AXOpen.Components.Abstractions.Drives.eAxoDriveDirection;         //  Enum type (1-of-4 values: PositiveDirection, ShortestWay, NegativeDirection, CurrentDirection)
            END_VAR
            VAR_OUTPUT
                Done            :   BOOL;                       // Commanded position finally reached
                Busy            :   BOOL;                       // The method is not finished and new output values are to be expected
                Active          :   BOOL;                       // Indicates that the method has control on the axis
                CommandAborted  :   BOOL;                       // ‘Command’ is aborted by another command
                Error           :   BOOL;                       // Signals that an error has occurred within the method
                ErrorID         :   DINT;                       // Error identification
            END_VAR
            VAR
                _AxisReference :  REF_TO AxoCtrlxDriveXscAxisReference;
            END_VAR

            _AxisReference ?= AxisRef;

            IF(_AxisReference = NULL) THEN
                Messenger.Activate(     UINT#1490, eAxoMessageCategory#ProgrammingError);
                DriveStatus.Error.Id := UINT#1490;
                RETURN;
            END_IF;

            IF THIS.AxoMoveAbsolute_Task.StartTriggered()  THEN
                _AxisReference^.Status.CurrentMotionTaskId := AXOpen.Components.Drives.eAxoMotionTaskId#Axo_MoveAbsolute;
            END_IF;

            IF Execute AND NOT MC_MoveAbsoluteExecute_PV AND _State = UINT#0 THEN
                _AxisReference^.Data.Cycle := _AxisReference^.Data.Cycle + ULINT#2;
                MC_MoveAbsoluteCycle := _AxisReference^.Data.Cycle ;
            END_IF;

            IF Execute THEN
                Messenger.ActivateOnCondition(ULINT#1491, Execute AND Velocity <= 0, eAxoMessageCategory#ProgrammingError);
                Messenger.ActivateOnCondition(ULINT#1492, Execute AND Acceleration <= 0, eAxoMessageCategory#ProgrammingError);
                Messenger.ActivateOnCondition(ULINT#1493, Execute AND Deceleration <= 0, eAxoMessageCategory#ProgrammingError);
                Messenger.ActivateOnCondition(ULINT#1494, Execute AND Jerk <= 0, eAxoMessageCategory#ProgrammingError);

                IF NOT ContinuousUpdate THEN
                    MC_MoveAbsoluteContinuousUpdate_SV := FALSE;
                END_IF;
                IF _State = UINT#0 THEN
                    Busy := TRUE;
                    Active := TRUE;
                    MC_MoveAbsoluteErrorID := DINT#0;
                    _AxisReference^.Outputs.SignalControlWord_S_0_0145_0_0.JogPositive      := FALSE;
                    _AxisReference^.Outputs.SignalControlWord_S_0_0145_0_0.JogNegative      := FALSE;
                    _AxisReference^.Outputs.SignalControlWord_S_0_0145_0_0.HomingControl    := FALSE;
                    _AxisReference^.Outputs.SignalControlWord_S_0_0145_0_0.AbsoluteRelative := FALSE;
                    MC_MoveAbsoluteContinuousUpdate_SV := ContinuousUpdate;
                    _State := UINT#350;
                    THIS.CallTimers(FALSE);
                END_IF;
                IF _State = UINT#350 THEN
                    IF _infoTimer.output THEN
                        TaskMessenger.Activate( UINT#550, eAxoMessageCategory#Potential);
                        DriveStatus.Error.Id := UINT#550;
                    END_IF;
                    Busy := TRUE;
                    Active := TRUE;
                    IF Velocity > 0 AND Acceleration > 0 AND Deceleration > 0 AND Jerk > 0 THEN
                        _AxisReference^.Outputs.CommandPosition_S_0_0282_0_0 :=         TO_DINT(Position        *   ScalingConstantRequiredPosition);
                        _AxisReference^.Outputs.CommandVelocity_S_0_0259_0_0 :=         TO_DINT(Velocity        *   ScalingConstantRequiredVelocity     * _AxisReference^.Data.OverrideVelocityFactor);
                        _AxisReference^.Outputs.CommandAcceleration_S_0_0260_0_0 :=     TO_DINT(Acceleration    *   ScalingConstantRequiredAcceleration * _AxisReference^.Data.OverrideAccelerationFactor);
                        _AxisReference^.Outputs.CommandDecceleration_S_0_0359_0_0 :=    TO_DINT(Deceleration    *   ScalingConstantRequiredDeceleration * _AxisReference^.Data.OverrideAccelerationFactor);
                        _AxisReference^.Outputs.CommandJerk_S_0_0193_0_0 :=             TO_DINT(Jerk            *   ScalingConstantRequiredJerk         * _AxisReference^.Data.OverrideJerkFactor);
                        MC_MoveAbsolutePosition_PV      :=  Position;
                        MC_MoveAbsoluteVelocity_PV      :=  Velocity;
                        MC_MoveAbsoluteAcceleration_PV  :=  Acceleration;
                        MC_MoveAbsoluteDeceleration_PV  :=  Deceleration;
                        MC_MoveAbsoluteJerk_PV          :=  Jerk;
                        MC_MoveAbsoluteDirection_PV     :=  Direction;
                        _State := UINT#351;
                        THIS.CallTimers(FALSE);
                    END_IF;
                END_IF;
                IF _State = UINT#351 THEN
                    IF _infoTimer.output THEN
                        TaskMessenger.Activate( UINT#551, eAxoMessageCategory#Potential);
                        DriveStatus.Error.Id := UINT#551;
                    END_IF;
                    Busy := TRUE;
                    Active := TRUE;
                    _AxisReference^.Outputs.DriveControlWord_S_0_0134_0_0.CommandOperationModeBit0  := FALSE;
                    _AxisReference^.Outputs.DriveControlWord_S_0_0134_0_0.CommandOperationModeBit1  := FALSE;
                    _AxisReference^.Outputs.DriveControlWord_S_0_0134_0_0.CommandOperationModeBit2  := FALSE;
                    IF  NOT _AxisReference^.Inputs.DriveStatusWord_S_0_0135_0_0.ActualOperatingModeBit0 AND
                        NOT _AxisReference^.Inputs.DriveStatusWord_S_0_0135_0_0.ActualOperatingModeBit1 AND
                        NOT _AxisReference^.Inputs.DriveStatusWord_S_0_0135_0_0.ActualOperatingModeBit2 THEN
                        _State := UINT#352;
                        THIS.CallTimers(FALSE);
                    END_IF;
                END_IF;
                IF _State = UINT#352 THEN
                    IF _infoTimer.output THEN
                        TaskMessenger.Activate( UINT#552, eAxoMessageCategory#Potential);
                        DriveStatus.Error.Id := UINT#552;
                    END_IF;
                    Busy := TRUE;
                    Active := TRUE;
                    IF  _AxisReference^.Inputs.DriveStatusWord_S_0_0135_0_0.ReadyForOperationBit0 AND
                        _AxisReference^.Inputs.DriveStatusWord_S_0_0135_0_0.ReadyForOperationBit1 THEN
                       _State := UINT#353;
                       THIS.CallTimers(FALSE);
                    END_IF;
                END_IF;
                IF _State = UINT#353 THEN
                    IF _infoTimer.output THEN
                        TaskMessenger.Activate( UINT#553, eAxoMessageCategory#Potential);
                        DriveStatus.Error.Id := UINT#553;
                    END_IF;
                    Busy := TRUE;
                    Active := TRUE;
                    _AxisReference^.Outputs.DriveControlWord_S_0_0134_0_0.DriveHalt  := TRUE;
                    IF _AxisReference^.Inputs.DriveStatusWord_S_0_0135_0_0.CommandProcessingStatus AND NOT _AxisReference^.Inputs.DriveStatusWord_S_0_0135_0_0.InStandstill  THEN
                       _State := UINT#354;
                       THIS.CallTimers(FALSE);
                    END_IF;
                END_IF;
                //Executing movement
                IF _State = UINT#354 THEN
                    IF _infoTimer.output THEN
                        TaskMessenger.Activate( UINT#554, eAxoMessageCategory#Potential);
                        DriveStatus.Error.Id := UINT#554;
                    END_IF;
                    Busy := TRUE;
                    Active := TRUE;
                    _AxisReference^.Outputs.SignalControlWord_S_0_0145_0_0.AcceptanceOfPositioningCommandValue := NOT _AxisReference^.Outputs.SignalControlWord_S_0_0145_0_0.AcceptanceOfPositioningCommandValue; // _AxisReference^.Outputs.SignalControlWord_S_0_0145_0_0.AcceptanceOfPositioningCommandValue := NOT _AxisReference^.Inputs.SignalStatusWord_S_0_0144_0_0.PositionCommandAck;
                    IF TRUE THEN
                        _State := UINT#355;
                        THIS.CallTimers(FALSE);
                    END_IF;
                END_IF;
                IF _State = UINT#355 THEN
                    IF _infoTimer.output THEN
                        TaskMessenger.Activate( UINT#555, eAxoMessageCategory#Potential);
                        DriveStatus.Error.Id := UINT#555;
                    END_IF;
                    Busy := TRUE;
                    Active := TRUE;
                    IF _AxisReference^.Outputs.SignalControlWord_S_0_0145_0_0.AcceptanceOfPositioningCommandValue = _AxisReference^.Inputs.SignalStatusWord_S_0_0144_0_0.PositionCommandAck THEN
                        _State := UINT#356;
                        THIS.CallTimers(FALSE);
                    END_IF;
                END_IF;
                IF _State = UINT#356 THEN
                    IF _infoTimer.output THEN
                        TaskMessenger.Activate( UINT#556, eAxoMessageCategory#Potential);
                        DriveStatus.Error.Id := UINT#556;
                    END_IF;
                    IF _AxisReference^.Inputs.SignalStatusWord_S_0_0144_0_0.DriveStandstill AND _AxisReference^.Inputs.SignalStatusWord_S_0_0144_0_0.InTargetPosition THEN
                        _State := UINT#357;
                        THIS.CallTimers(FALSE);
                    END_IF;
                END_IF;
                IF _State = UINT#357 THEN
                    Done := TRUE;
                    MC_MoveAbsoluteCycle := ULINT#0;
                END_IF;
                IF _State = UINT#358 THEN
                    CommandAborted := TRUE; // action handled in parent AxoDrive
                END_IF;
                IF _State = UINT#359 THEN
                    MC_MoveAbsoluteCycle := ULINT#0;
                    Error := TRUE; // action handled in parent AxoDrive
                END_IF;

                IF _State>=UINT#350 AND _State<UINT#357 THEN
                    IF MC_MoveAbsoluteContinuousUpdate_SV AND (
                        MC_MoveAbsolutePosition_PV      <>  Position OR
                        MC_MoveAbsoluteVelocity_PV      <>  Velocity OR
                        MC_MoveAbsoluteAcceleration_PV  <>  Acceleration OR
                        MC_MoveAbsoluteDeceleration_PV  <>  Deceleration OR
                        MC_MoveAbsoluteJerk_PV          <>  Jerk OR
                        MC_MoveAbsoluteDirection_PV     <>  Direction ) THEN
                        IF TRUE THEN
                            _State := UINT#350;
                        END_IF;
                    END_IF;
                    IF NOT _AxisReference^.Inputs.DriveStatusWord_S_0_0135_0_0.ReadyForOperationBit0 OR NOT _AxisReference^.Inputs.DriveStatusWord_S_0_0135_0_0.ReadyForOperationBit1 THEN
                        _State := UINT#358;
                    ELSIF _AxisReference^.Inputs.DriveStatusWord_S_0_0135_0_0.DriveErrorZKL1 OR
                        (_AxisReference^.Inputs.DriveStatusWord_S_0_0135_0_0.WarningZKL2 AND _AxisReference^.Inputs.DiagnosticMessage_S_0_0390_0_0 >= DWORD#16#C00E0000) THEN
                        // _debugCounter := _debugCounter + ULINT#1;
                        IF MC_MoveAbsoluteErrorID = DINT#0 THEN
                            MC_MoveAbsoluteErrorID := TO_DINT(_AxisReference^.Inputs.DiagnosticMessage_S_0_0390_0_0 AND DWORD#16#000FFFFF);
                        END_IF;
                        _State := UINT#359;
                    ELSIF _AxisReference^.Data.Cycle <> MC_MoveAbsoluteCycle THEN
                        _AxisReference^.Data.Cycle := _AxisReference^.Data.Cycle - ULINT#1;
                        _State := UINT#358;
                    END_IF;
                END_IF;

                THIS.CallTimers(TRUE,FALSE);
                THIS.AxoMoveAbsolute_Task.ThrowWhen(_errorTimer.output );
                THIS.AxoMoveAbsolute_Task.ThrowWhen(THIS.AxoMoveAbsolute_Task.Duration >= DriveConfig.TaskTimeout AND DriveConfig.TaskTimeout > T#0s ,'<#AxoMoveAbsolute_Task timeout.#>');
                DriveStatus.Action.Id := _State;
            END_IF;

            IF THIS.AxoMoveAbsolute_Task.DoneReached() AND _State>=UINT#350 AND _State<=UINT#359 THEN
                _AxisReference^.Status.CurrentMotionTaskId := AXOpen.Components.Drives.eAxoMotionTaskId#Axo_Done;
                MC_MoveAbsoluteErrorID := DINT#0;
                _State := UINT#0;
            END_IF;

            IF THIS.AxoMoveAbsolute_Task.RestoreTriggered() AND _State>=UINT#350 AND _State<=UINT#359 THEN
                _AxisReference^.Status.CurrentMotionTaskId := AXOpen.Components.Drives.eAxoMotionTaskId#Axo_None;
                MC_MoveAbsoluteErrorID := DINT#0;
                MC_MoveAbsoluteCycle := ULINT#0;
                _State := UINT#0;
                MC_MoveAbsoluteExecute_PV := FALSE;
            END_IF;
            ErrorID := MC_MoveAbsoluteErrorID;
            MC_MoveAbsoluteExecute_PV := Execute;
        END_METHOD
